(* IEC 61131-3 sources: mastertool-rankine-bridge/tests/indexer/fixtures/sample_export/objects/application_fb_0__FB_ValvulaSintetica, 1 file *)

(* ---- declaration.st ---- *)
FUNCTION_BLOCK FB_ValvulaSintetica
VAR_INPUT
    xComandoAbrir   : BOOL;
    tTempoLimite    : TIME := T#2S;
END_VAR
VAR_OUTPUT
    xValvulaAberta  : BOOL;
    xFalhaValvula   : BOOL;
END_VAR
VAR
    tonMonitorAbre  : TON;
END_VAR
VAR CONSTANT
    iMaxTentativas  : INT := 3;
END_VAR
